FUNCTION_BLOCK AMP4220 
VAR_INPUT
END_VAR
VAR_OUTPUT
	
			MoverTypeWidth 				: 		LREAL := 56.5; // Mover Width/2 in mm
			MoverTypeLength				: 		LREAL := 56.5; // Mover Length/2 in mm 

END_VAR
VAR
END_VAR

END_FUNCTION_BLOCK

(* stored: Version 1.1.0.1, ProductVersion 3.1.4024.12
   POU AMP4220: Id {53faabf0-435f-451c-bfbb-05458eef97df}, SpecialFunc None *)
